FUNCTION_BLOCK FB_TABLE (* Abstract superclass for HMI elements containing a table. *)
  (* Standard: 61499-2 *)
  (* Version 0.0, 2004-06-22, JHC, Rockwell Automation *)
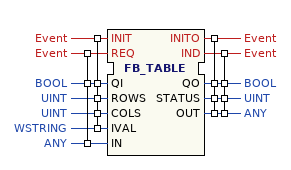
  EVENT_INPUT
    INIT WITH QI, ROWS, COLS, IVAL; (* Initialize matrix to IN *)
    REQ WITH QI, IN; (* Set table values(for table outputs only) *)
  END_EVENT
  EVENT_OUTPUT
    INITO WITH QO, STATUS, OUT; (* Initialization Confirm *)
    IND WITH QO, STATUS, OUT; (* Confirmation of REQ(for table outputs)or user inputs(for table inputs) *)
  END_EVENT
  VAR_INPUT
    QI : BOOL; (* 1=Enabled,0=Inhibited *)
    ROWS : UINT := 1; (* Number of rows in the table *)
    COLS : UINT := 1; (* Number of columns in the table *)
    IVAL : WSTRING; (* Initialization string(subclass-dependent) *)
    IN : ANY; (* Data to update table(implementation-dependent) *)
  END_VAR
  VAR_OUTPUT
    QO : BOOL; (* 0=OK,1=Inhibited *)
    STATUS : UINT; (* 0=OK,2=TYPE_CONVERSION_ERROR,4=INHIBITED,13=ARRAY_SIZE_ERROR *)
    OUT : ANY; (* Output data from table(implementation-dependent) *)
  END_VAR
  SERVICE FB_TABLE/table
    SEQUENCE normal_initialization
      FB_TABLE.INIT+(ROWS,COLS,IVAL) -> table.initialize() -> FB_TABLE.INITO+(OUT);
    END_SEQUENCE
    SEQUENCE unsuccessful_initialization
      FB_TABLE.INIT+(ROWS,COLS,IVAL) -> table.initialize() -> FB_TABLE.INITO-(STATUS);
    END_SEQUENCE
    SEQUENCE initialization_inhibited
      FB_TABLE.INIT-() -> FB_TABLE.INITO-(STATUS);
    END_SEQUENCE
    SEQUENCE request
      FB_TABLE.REQ+(IN) -> table.update() -> FB_TABLE.IND+(OUT);
    END_SEQUENCE
    SEQUENCE request_inhibited
      FB_TABLE.REQ-() -> FB_TABLE.IND-(STATUS);
    END_SEQUENCE
    SEQUENCE table_not_initialized
      FB_TABLE.REQ+(IN) -> FB_TABLE.IND-(STATUS);
    END_SEQUENCE
    SEQUENCE request_error
      FB_TABLE.REQ+(IN) -> table.request() -> FB_TABLE.CNF-(STATUS);
    END_SEQUENCE
    SEQUENCE user_input
      table.setValue() -> FB_TABLE.IND+(OUT);
    END_SEQUENCE
    SEQUENCE user_input_inhibited
      table.setValue(QI=FALSE);
    END_SEQUENCE
    SEQUENCE user_input_error
      table.setValue();
    END_SEQUENCE
  END_SERVICE
END_FUNCTION_BLOCK
